PROGRAM MAIN
VAR
	selectedIndex: INT := 0;
	px: MotorProxy;
	motors: ARRAY[0..3] OF Motor;
	
	
	aComboboxEntries : ARRAY [0..5] OF ST_ComboboxEntry;

	
	
	
END_VAR


	aComboboxEntries[0].id:=0;
	aComboboxEntries[0].text:="Motor One";
	aComboboxEntries[0].value:=0;
	
	
	






//	GVL.motors[0].name := "One";
	motors[0].motorId := 1;
	motors[0].isAxisSelected := 1;
	motors[0].encoder := 0.012;
	motors[0].status := AxisStatus.Ready;
	
	//GVL.motors[1].name := "Two";
	motors[1].motorId := 2;
	motors[1].isAxisSelected := 1;
	motors[1].encoder := 0.012;
	motors[1].status := AxisStatus.Ready;
	
	//GVL.motors[2].name := "Three";
	motors[2].motorId := 3;
	motors[2].isAxisSelected := 1;
	motors[2].encoder := 0.012;
	motors[2].status := AxisStatus.Ready;

END_PROGRAM

(* stored: Version 1.1.0.1, ProductVersion 3.1.4024.13
   POU MAIN: Id {d8b28e72-1144-429e-a297-29a2c3b328e4}, SpecialFunc None *)
